TYPE Udt_CM_Sensor2State :
STRUCT
	PI_ManualMode : BOOL;
	PI_AutoHigh : BOOL;
	
	PI_HMI_HAND : BOOL;
	PI_HMI_HAND_ON : BOOL;
	
	PI_AlarmHighEnable : BOOL;
	PI_AlarmLowEnable : BOOL;
	
	PI_Alarmdelay_H : INT;
	PI_Alarmdelay_L : INT;
	
	PO_Alarm_H : BOOL;
	PO_Alarm_L : BOOL;
	
	PO_HMI_HAND : BOOL;
	PO_High : BOOL;
	
	PO_HIST_BIT_H : BOOL;
	PO_HIST_BIT_L : BOOL;

END_STRUCT
END_TYPE

(* stored: Version 1.1.0.1, ProductVersion 3.1.4024.13
   DUT Udt_CM_Sensor2State: Id {2f6388ed-cb02-4321-a41b-1485be11ae1f} *)
